TYPE ST_DeviceDiagnosticsStatus :
STRUCT
    bCriticalDeviceFault        : BOOL;
END_STRUCT
END_TYPE

(* stored: Version 1.1.0.1, ProductVersion 3.1.4024.16
   DUT ST_DeviceDiagnosticsStatus: Id {f9c23e54-f6ae-40cf-af9c-faa6b364c88e} *)
